(* CODESYS project WaschMa.export

Project tree, tasks and I/O mapping:
  Device : CODESYS Control for PFC200 SL, CODESYS, order no. 2302000010, version 4.15.0.0
    application Application
      libraries: Standard, 3.5.18.0 (System)
      task MainTask (cyclic, interval t#20ms, priority 1) calls PLC_PRG
      program PLC_PRG [ST]
    A1_WaschMa : Wago PFC100 interner Bus, CODESYS, version 4.19.0.0
      A2_DI : 750-1415 8DI, WAGO Kontakttechnik GmbH u. Co. KG, order no. 750-1415, version 4.19.0.0
          input  S0_NotHalt : BOOL  // Digital Inputs 0 - 7.DI0
          input  S1_ProgrammWahl_1 : BOOL  // Digital Inputs 0 - 7.DI1
          input  S1_ProgrammWahl_2 : BOOL  // Digital Inputs 0 - 7.DI2
          input  S1_ProgrammWahl_3 : BOOL  // Digital Inputs 0 - 7.DI3
          input  S3_DeckelGechlossen : BOOL  // Digital Inputs 0 - 7.DI4
          input  S11_WasserstandHigh : BOOL  // Digital Inputs 0 - 7.DI5
          input  S10_WasserstandLow : BOOL  // Digital Inputs 0 - 7.DI6
          unmapped channels: Digital Inputs 0 - 7
      A3_DI : 750-1415 8DI, WAGO Kontakttechnik GmbH u. Co. KG, order no. 750-1415, version 4.19.0.0
          unmapped channels: Digital Inputs 0 - 7
      A4_DO : 750-1515 8DO, WAGO Kontakttechnik GmbH u. Co. KG, order no. 750-1515, version 4.19.0.0
          output V1_Wasser : BOOL  // Digital Outputs 0 - 7.DO0
          output V2_Waschmittel : BOOL  // Digital Outputs 0 - 7.DO1
          output V3_Weichspueler : BOOL  // Digital Outputs 0 - 7.DO2
          output V4_Abwasser : BOOL  // Digital Outputs 0 - 7.DO3
          output K1_Heizung : BOOL  // Digital Outputs 0 - 7.DO4
          output M2_Abwasser : BOOL  // Digital Outputs 0 - 7.DO5
          unmapped channels: Digital Outputs 0 - 7
      A5_DO : 750-1515 8DO, WAGO Kontakttechnik GmbH u. Co. KG, order no. 750-1515, version 4.19.0.0
          output U1_Freigabe : BOOL  // Digital Outputs 0 - 7.DO0
          output U1_Drehrichtung : BOOL  // Digital Outputs 0 - 7.DO1
          output U1_Start : BOOL  // Digital Outputs 0 - 7.DO2
          unmapped channels: Digital Outputs 0 - 7
      A6_RTD : 750-450 4AI, RTD, WAGO Kontakttechnik GmbH u. Co. KG, order no. 750-450, version 4.19.0.0
          unmapped channels: Analog Input Channel 0, Analog Input Channel 1, Analog Input Channel 2, Analog Input Channel 3
      A7_AI : 75x-455 4AE, 4-20 mA, WAGO Kontakttechnik GmbH & Co. KG, order no. 75x-455, version 4.19.0.0
          input  U1_IstDrehzahl : INT  // Analog Input Channel 0
          unmapped channels: Analog Input Channel 1, Analog Input Channel 2, Analog Input Channel 3
      A8_AO : 75x-553 4AO, 0-20 mA, WAGO Kontakttechnik GmbH u. Co. KG, order no. 75x-553, version 4.19.0.0
          output U1_SollDrehzahl : INT  // Analog Output Channel 0
          unmapped channels: Analog Output Channel 1, Analog Output Channel 2, Analog Output Channel 3
*)

// Device/Application/PLC_PRG
PROGRAM PLC_PRG
VAR
	bProgrammWahl_1 :BOOL;
	bProgrammWahl_2 :BOOL;
	bProgrammWahl_3 :BOOL;
END_VAR


 IF S0_NotHalt THEN
	 ;
 	bProgrammwahl_1 := S1_ProgrammWahl_1;
	bProgrammwahl_2 := S1_ProgrammWahl_2;
	bProgrammwahl_3 := S1_ProgrammWahl_3;      
 ELSE
	 
 	V1_Wasser        := FALSE;
	V2_Waschmittel   := FALSE;
	V3_Weichspueler  := FALSE;
	V4_Abwasser 	 := FALSE;
	K1_Heizung 		 := FALSE;
	M2_Abwasser 	 := FALSE;
	U1_Freigabe    	 := FALSE;
	U1_Start         := FALSE;
	U1_SollDrehzahl  := 0;
	
 END_IF

END_PROGRAM
